(* IEC 61131-3 sources: ECU_Test_Arduino_PLC/PLC_Software, 6 files *)

(* ---- GVL.ST ---- *)
{attribute 'qualified_only'}
VAR_GLOBAL CONSTANT
	uiPeriodcMessageN : UINT := 2;
	uiRXMessageN : UINT := 3;
END_VAR

VAR_GLOBAL
	aPeriodicMessages: ARRAY[1..GVL.uiPeriodcMessageN] OF PERIODIC_MESSAGE;
	aRXMessages: ARRAY[1..GVL.uiRXMessageN] OF RX_MESSAGE;

END_VAR

(* ---- GVL_IO.ST ---- *)
{attribute 'qualified_only'}
VAR_GLOBAL
	//w_CAN_SEND: ARRAY[0..23] OF BYTE;
	//AUX IO
	x_PEDAL_REAL: BOOL;
	x_PEDAL_TYPE: BOOL;

	x_DOG12 : BOOL	;//	J1.E1	Red Changing Light
	x_DOG01	: BOOL	;//	J1.E2	Contactor Supply Control Packs 4-6
	x_DOG02	: BOOL	;//	J1.E3	Contactor Supply Control Packs 7-9
	x_DOG03	: BOOL	;//	J1.E4	Start/Stop Orange LED
	x_DOG04	: BOOL	;//	J1.F1	Start/Stop Green LED
	x_DOG05	: BOOL	;//	J1.F2	Green Charging Light
	x_DOG06	: BOOL	;//	J1.F3 	Contactor Supply Control Packs 1-3
	x_DOG07	: BOOL	;//	J1.F4 	Blue Charging Light
	x_DOG08	: BOOL	;//	J1.G1 	TGC Off Command
	x_DOG09	: BOOL	;//	J1.G2 	TGC On Command
	x_DOG10	: BOOL	;//	J1.G3	LV ePTO Relay Coil control
	x_DOG11	: BOOL	;//	J1.G4	Differential Lock Solenoid LS

	x_DOV01	: BOOL	;//	J1.L1	VCM Wake 1
	x_DOV02	: BOOL	;//	J1.L2	VCM Wake 2
	x_DOV03	: BOOL	;//	J1.L3	VCM Wake 3
	x_DOV04	: BOOL	;//	J1.L4	Governor Valve
	x_DOV05	: BOOL	;//	J1.M1	Regeneration Valve
	x_DOV06	: BOOL	;//	J1.M2	VCM wake 4
	x_DOV07	: BOOL	;//	J1.M3	Auxiliary HVIL Out
	x_DOV08	: BOOL	;//	J1.M4	HV Battery 1-9 Wake

	x_DHLC01 : BOOL	;// J3.21 Cabin Tilt Status [Digital HS-LS Control 1]
	x_DFC01	 : BOOL; // J3.21 Cabin Tilt Status [Digital Float Control 1]
	x_DHLC02 : BOOL	;// J3.22 Drive Req Signal 1 [Digital HS-LS Control 2]
	x_DFC02	 : BOOL; // J3.22 Drive Req Signal 1 [Digital Float Control 2]
	x_DHLC03 : BOOL	;// J3.33 Drive Req Signal 2 [Digital HS-LS Control 3]
	x_DFC03	 : BOOL; // J3.33 Drive Req Signal 2 [Digital Float Control 3]
	x_DHLC04 : BOOL	;// J3.34 Neutral Req Signal [Digital HS-LS Control 4]
	x_DFC04	 : BOOL; // J3.34 Neutral Req Signal [Digital Float Control 4]
	x_DHLC05 : BOOL	;// J3.45 Reverse Req Signal 1 [Digital HS-LS Control 5]
	x_DFC05	 : BOOL; // J3.45 Reverse Req Signal 1 [Digital Float Control 5]
	x_DHLC06 : BOOL	;// J3.46 Reverse Req Signal 2 [Digital HS-LS Control 6]
	x_DFC06	 : BOOL ; // J3.46 Reverse Req Signal 2 [Digital Float Control 6]

	x_CF01	 : BOOL ; // J3.23 Start/Stop Signal 2 [Control Float 1]
	x_CF02	 : BOOL ; // J3.24 Start/Stop Signal 1 [Control Float 2]
	x_CF03	 : BOOL ; // J3.25 APU Sensor Front Signal [Control Float 3]
	x_CF04	 : BOOL ; // J3.26 APU Sensor Rear Signal [Control Float 4]
	x_CF05	 : BOOL ; // J3.27 TGC Off Request [Control Float 5]
	x_CF06	 : BOOL ; // J3.28 TGC On Request [Control Float 6]
	x_CF07	 : BOOL ; // J3.35 FLEX-IN6 [Control Float 7]
	x_CF08	 : BOOL ; // J3.36 FLEX-IN7 [Control Float 8]
	x_CF09	 : BOOL ; // J3.37 FLEX-IN8 [Control Float 9]
	x_CF10	 : BOOL ; // J3.38 Positive Auxiliary Contactor Feedback [Control Float 10]
	x_CF11	 : BOOL ; // J3.39 Negative Auxiliary Contactor Feedback [Control Float 11]
	x_CF12	 : BOOL ; // J3.40 FLEX-IN11 [Control Float 12]
	x_CF13	 : BOOL ; // J3.47 HW E-Stop Signal [Control Float 13]
	x_CF14	 : BOOL ; // J3.48 TPMS Power [Control Float 14]
	x_CF15	 : BOOL ; // J3.49  Differential Lock Sensor Signal [Control Float 15]
	x_CF16	 : BOOL ; // J3.50  Charge Door Position [Control Float 16]

	x_CA01	 : BOOL ; // J3.23 Start/Stop Signal 2 [Control Analog 1]
	x_CA02	 : BOOL ; // J3.24 Start/Stop Signal 1 [Control Analog 2]
	x_CA03	 : BOOL ; // J3.25 APU Sensor Front Signal [Control Analog 3]
	x_CA04	 : BOOL ; // J3.26 APU Sensor Rear Signal [Control Analog 4]
	x_CA05	 : BOOL ; // J3.27 TGC Off Request [Control Analog 5]
	x_CA06	 : BOOL ; // J3.28 TGC On Request [Control Analog 6]
	x_CA07	 : BOOL ; // J3.35 FLEX-IN6 [Control Analog 7]
	x_CA08	 : BOOL ; // J3.36 FLEX-IN7 [Control Analog 8]
	x_CA09	 : BOOL ; // J3.37 FLEX-IN8 [Control Analog 9]
	x_CA10	 : BOOL ; // J3.38 Positive Auxiliary Contactor Feedback [Control Analog 10]
	x_CA11	 : BOOL ; // J3.39 Negative Auxiliary Contactor Feedback [Control Analog 11]
	x_CA12	 : BOOL ; // J3.40 FLEX-IN11 [Control Analog 12]
	x_CA13	 : BOOL ; // J3.47 HW E-Stop Signal [Control Analog 13]
	x_CA14	 : BOOL ; // J3.48 TPMS Power [Control Analog 14]
	x_CA15	 : BOOL ; // J3.49  Differential Lock Sensor Signal [Control Analog 15]
	x_CA16	 : BOOL ; // J3.50  Charge Door Position [Control Analog 16]

	w_FlexIN0	 : WORD ; // J3.23 Start/Stop Signal 2 [FlexIN0]
	w_FlexIN1	 : WORD ; // J3.24 Start/Stop Signal 1 [FlexIN1]
	w_FlexIN2	 : WORD ; // J3.25 APU Sensor Front Signal [FlexIN2]
	w_FlexIN3	 : WORD ; // J3.26 APU Sensor Rear Signal [FlexIN3]
	w_FlexIN4	 : WORD ; // J3.27 TGC Off Request [FlexIN4]
	w_FlexIN5	 : WORD ; // J3.28 TGC On Request [FlexIN5]
	w_FlexIN6	 : WORD ; // J3.35 FLEX-IN6 [FlexIN6]
	w_FlexIN7	 : WORD ; // J3.36 FLEX-IN7 [FlexIN7]
	w_FlexIN8	 : WORD ; // J3.37 FLEX-IN8 [FlexIN8]
	w_FlexIN9	 : WORD ; // J3.38 Positive Auxiliary Contactor Feedback [FlexIN9]
	w_FlexIN10	 : WORD ; // J3.39 Negative Auxiliary Contactor Feedback [FlexIN10]
	w_FlexIN11	 : WORD ; // J3.40 FLEX-IN11 [FlexIN11]
	w_FlexIN12	 : WORD ; // J3.47 HW E-Stop Signal [FlexIN12]
	w_FlexIN13	 : WORD ; // J3.48 TPMS Power [FlexIN13]
	w_FlexIN14	 : WORD ; // J3.49  Differential Lock Sensor Signal [FlexIN14]
	w_FlexIN15	 : WORD ; // J3.50  Charge Door Position [FlexIN15]

	w_AccPedalSig1			: WORD 	;	//J3.8 AccPedalSig1
	w_AccPedalSig2			: WORD  ;	//J3.9 AccPedalSig2
	w_ANC2					: WORD  ;	//J3.10 ANC2
	w_OilLevelSig			: WORD  ;	//J3.11 OilLevelSig
	w_Cabin_Sw_E_Stop_Sig	: WORD  ;	//J3.12 Cabin_Sw_E_Stop_Sig
	w_ANC5					: WORD  ;	//J3.13 ANC5

	b_PWM1_Control_Byte_0	: BYTE ;   // J3.19-20 PWM [Control Byte 0]
	w_PWM1_DO1				: WORD ;   // J3.19 Speed Pulse PWM [DO1]
	w_PWM1_DO2				: WORD ;   // J3.20 Distance Signal [DO2]
	b_PWM1_Control_Byte_2   : BYTE ;  // J3.31-32 PWM [Control Byte 2]
	w_PWM1_DO3				: WORD ;   // J3.31 FLEX_PWM2_NOT_USED [DO3]
	w_PWM1_DO4				: WORD ;   // J3.32 PYRO Crash Event Signal [DO4]

	b_PWM2_Control_Byte_0	: BYTE ;   // J3.43-44 PWM [Control Byte 0]
	w_PWM2_DO1				: WORD ;   // J3.43 FLEX_PWM4 [DO1]
	w_PWM2_DO2				: WORD ;   // J3.44 FLEX_PWM5 [DO2]

//	x_DOV09	: BOOL	;//	X2.28	b
//	x_CrankHSS	: BOOL	;//	X2.36	Cranking Relay HSS
//	x_DOV15	: BOOL	;//	X2.06	Single H out2
//	x_DOV16	: BOOL	;//	X2.04	Single H out1
	//LIN1-GND	: BOOL	;//	X1.05	LIN 1 GND
	x_TRX_P	: BOOL	;//	X1.07	Not Used
	x_TRX_M	: BOOL	;//	X1.08	Not Used
	//x_DIG_ACC_GND: BOOL	;//	X1.09	Accelerator pedal low idle switch
	//x_DIG16	: BOOL	;//	X1.10	PTO 3
	//x_DIG15	: BOOL	;//	X1.11	PTO 2
	//x_DIG14	: BOOL	;//	X1.12	PTO 1
	x_DIB15	: BOOL	;//	X1.13	Hill holder
	x_DIB15H	: BOOL	;//	X1.13	Hill holder
	//LIN2-GND	: BOOL	;//	X1.14	optional
	x_ASG02	: BOOL	;//	X1.15	Accelerator Pedal channel2 Ground
	//CAN6-H	: BOOL	;//	X1.16	Not Used
	//CAN6-L	: BOOL	;//	X1.17	Not Used
	x_ASG01	: BOOL	;//	X1.18	Accelerator Pedal channel1 Ground
	//CAN5-H	: BOOL	;//	X1.19	Body Computer Bus - CAN H
	//CAN5-L	: BOOL	;//	X1.20	Body Computer Bus - CAN L
	w_AI01	: WORD	;//	X1.21	Accelerator Pedal channel 1
	w_AI02	: WORD	;//	X1.22	Accelerator Pedal channel 2
	x_ACC_SW_GND: BOOL	;//	X1.23	Accelerator  pedal low idle switch Ground

	x_ASV01	: BOOL	;//	X1.26	Accelerator Pedal channel 1 Supply
	x_ASV02	: BOOL	;//	X1.27	Accelerator Pedal channel 2 Supply
	x_AWWS_B_In	: BOOL	;//	X1.28	optional
	x_AWWS_B_Out: BOOL	;//	X1.29	optional
	//LIN1-SIG	: BOOL	;//	X1.31	LIN 1 Bus
	//LIN2-SIG	: BOOL	;//	X1.32	optional
	//LIN1-SUP	: BOOL	;//	X1.33	LIN 1 supply
	//LIN2-SUP	: BOOL	;//	X1.34	optional
	x_AWWS_A_In	: BOOL	;//	X1.35	optional
	x_AWWS_A_Out: BOOL	;//	X1.36	optional

	x_TRM_30: BOOL	;//	X2.01	Power Supply
	//CAN9-H	: BOOL	;//	X2.02	optional
	//CAN9-L	: BOOL	;//	X2.03	optional

	x_AI03	: BOOL	;//	X2.07	Analog Input 3
	//x_DIG07	: BOOL	;//	X2.08	Gear High/Low
	x_TRM_15: BOOL	;//	X2.09	Ignition Key
	//CAN1-H	: BOOL	;//	X2.10	Vehicle Data Bus CAN H
	//CAN1-L	: BOOL	;//	X2.11	Vehicle Data Bus CAN L
	//CAN2-H	: BOOL	;//	X2.12	Engine Contro Bus - CAN H
	//CAN2-L	: BOOL	;//	X2.13	Engine Contro Bus - CAN L
	//CAN3-H	: BOOL	;//	X2.14	Expansion Module Bus - CAN H
	//CAN3-L	: BOOL	;//	X2.15	Expansion Module Bus - CAN L
	//CAN4-H	: BOOL	;//	X2.16	ADAS Data Bus CAN FD - CAN H
	//CAN4-L	: BOOL	;//	X2.17	ADAS Data Bus CAN FD - CAN L
	x_TRM_31: BOOL	;//	X2.19	Power Supply GND
	x_DIV04	: BOOL	;//	X2.20	Alcohol Interlock
	//x_DIG12	: BOOL	;//	X2.21	BB Start
	//x_DIG13	: BOOL	;//	X2.22	BB Stop
	//cAN7-H	: BOOL	;//	X2.23	optional
	//CAN7-L	: BOOL	;//	X2.24	optional
	//CAN8-H	: BOOL	;//	X2.25	optional
	//CAN8-L	: BOOL	;//	X2.26	optional

	x_DIB16	: BOOL	;//	X2.30	Halt brake
	x_DIB16H: BOOL	;//	X2.30	Halt brake
	x_DIB17	: BOOL	;//	X2.31	ESP / ASR
	x_DIB17H: BOOL	;//	X2.31	ESP / ASR

	//x_DIG19	: BOOL	;//	X2.34	Clima 22
	//x_DIG18	: BOOL	;//	X2.35	Clima 18

// 	x_DIG01	: BOOL	;//	X3.01	CC Set+
// 	x_DIG02	: BOOL	;//	X3.02	CC Set-
// 	x_DIG03	: BOOL	;//	X3.03	CC Resume
// 	x_DIG04	: BOOL	;//	X3.04	CC Off
	x_DIB05	: BOOL	;//	X3.05	CC GAP-
	x_DIB05H: BOOL	;//	X3.05	CC GAP-
	x_DIB06	: BOOL	;//	X3.06	CC GAP +
	x_DIB06H: BOOL	;//	X3.06	CC GAP +
// 	x_DIG05	: BOOL	;//	X3.07	Ext/Int CC
// 	x_DIG20	: BOOL	;//	X3.08	D/Dm1
// 	x_DIG24	: BOOL	;//	X3.09	R/Rm1
// 	x_DIG22	: BOOL	;//	X3.10	N
// 	x_DIG21	: BOOL	;//	X3.11	D/Dm2
// 	x_DIG25	: BOOL	;//	X3.12	R/Rm2
	x_DIB12	: BOOL	;//	X3.13	Gear Up
	x_DIB12H	: BOOL	;//	X3.13	Gear Up
	x_DIB13	: BOOL	;//	X3.14	Gear Down
	x_DIB13H	: BOOL	;//	X3.14	Gear Down
	x_DIB04	: BOOL	;//	X3.15	FPSL
	x_DIB04H	: BOOL	;//	X3.15	FPSL
	x_DIB02	: BOOL	;//	X3.16	ECO Roll Swt
	x_DIB02H	: BOOL	;//	X3.16	ECO Roll Swt
	x_DIV03	: BOOL	;//	X3.17	Second SL Switch
	x_DIV02	: BOOL	;//	X3.18	Sec. Brake
	x_DIV01	: BOOL	;//	X3.19	Prim. Brake
	x_DIB11	: BOOL	;//	X3.20	ACC
	x_DIB11H	: BOOL	;//	X3.20	ACC
	x_DIB08	: BOOL	;//	X3.21	PECC
	x_DIB08H	: BOOL	;//	X3.21	PECC
	x_DIB01	: BOOL	;//	X3.22	Cranck request (K50)
	x_DIB01H	: BOOL	;//	X3.22	Cranck request (K50)
	x_DIB14	: BOOL	;//	X3.23	Parking Brake Switch
	x_DIB14H	: BOOL	;//	X3.23	Parking Brake Switch
	x_DIG11	: BOOL	;//	X3.24	Cabin Tilt
	x_DIG10	: BOOL	;//	X3.25	Neutral
	x_DIG06	: BOOL	;//	X3.26	Clutch
	//x_DIG17	: BOOL	;//	X3.27	Clutch 2nd
	x_DIB10	: BOOL	;//	X3.28	ABS OFF
	x_DIB10H	: BOOL	;//	X3.28	ABS OFF
	//x_DIG09	: BOOL	;//	X3.29	EB Mode 1
	x_DIB07	: BOOL	;//	X3.30	EB request
	x_DIB07H	: BOOL	;//	X3.30	EB request
	//x_DIG27	: BOOL	;//	X3.31	CSF - LDWS
	//x_DIG23	: BOOL	;//	X3.32	Heavy Offroad
	x_DIB03	: BOOL	;//	X3.33	Rocking Mode
	x_DIB03H	: BOOL	;//	X3.33	Rocking Mode
	x_DIB09	: BOOL	;//	X3.34	 Power mode
	x_DIB09H	: BOOL	;//	X3.34	 Power mode
	//x_DIG26	: BOOL	;//	X3.35	Silent Mode
	//x_DIG08	: BOOL	;//	X3.36	ECO Mode
END_VAR

(* ---- FB_RXCanMessageelaboration.ST ---- *)
FUNCTION_BLOCK FB_RXCanMessageElaboration
VAR_INPUT
	wRxId:WORD;
	bRxNBytes:BYTE;
	aRxBuffer: ARRAY [0..7] OF BYTE;
END_VAR
VAR_OUTPUT
END_VAR
VAR
	_FbCanTx11BitFrame : FbCanTx11BitFrame;
	xCANTxTrigger : BOOL;
	lut1,lut2: LUT;
END_VAR

xCANTxTrigger := FALSE;//no answer required

CASE wRxId OF
// 	16#75C:
// 			//ON MESSAGE ACTION
// 			IF aRxBuffer[0] = 0 THEN
// 				GVL.DO01 := FALSE;
// 			ELSE
// 				GVL.DO01 := TRUE;
// 			END_IF
// 			xCANTxTrigger := TRUE;
	16#11://BANCO_VCM4_Command
			GVL_IO.x_PEDAL_TYPE := aRxBuffer[0].0;//Pedal_Type
			GVL_IO.x_TRM_30 := aRxBuffer[0].1;//Power_Supply
			GVL_IO.x_TRM_15 := aRxBuffer[0].2;//Ignition_Key
			GVL_IO.x_PEDAL_REAL	:= aRxBuffer[0].3;//Accelerator_Pedal

	16#12://BANCO_VCM4_ANALOG_Critical_ADC (597_3) ++
			//ON MESSAGE ACTION
			GVL_IO.w_AccPedalSig1 := INT_TO_WORD(REAL_TO_INT((WORD_TO_REAL(SHL(BYTE_TO_WORD(aRxBuffer[1]),8) + BYTE_TO_WORD(aRxBuffer[0]))) * 0.001 * 32767) ); // Refer to the manual of 597 page 34
			GVL_IO.w_AccPedalSig2 := INT_TO_WORD(REAL_TO_INT((WORD_TO_REAL(SHL(BYTE_TO_WORD(aRxBuffer[3]),8) + BYTE_TO_WORD(aRxBuffer[2]))) * 0.001 * 32767) ); // Refer to the manual of 597 page 34
			GVL_IO.w_OilLevelSig := INT_TO_WORD(REAL_TO_INT((WORD_TO_REAL(SHL(BYTE_TO_WORD(aRxBuffer[5]),8) + BYTE_TO_WORD(aRxBuffer[4]))) * 0.001 * 32767) ); // Refer to the manual of 597 page 34
			GVL_IO.w_Cabin_Sw_E_Stop_Sig := INT_TO_WORD(REAL_TO_INT((WORD_TO_REAL(SHL(BYTE_TO_WORD(aRxBuffer[7]),8) + BYTE_TO_WORD(aRxBuffer[6]))) * 0.001 * 32767) ); // Refer to the manual of 597 page 34

	16#14://BANCO_VCM4_DI ++
			GVL_IO.x_DHLC01 := aRxBuffer[0].0; // Cabin_Tilt_Status_HS_LS
			GVL_IO.x_DFC01  := aRxBuffer[0].1; // Cabin_Tilt_Status_Float
			GVL_IO.x_DHLC02 := aRxBuffer[0].2; // Drive_Req_Signal_1_HS_LS
			GVL_IO.x_DFC02  := aRxBuffer[0].3; // Drive_Req_Signal_1_Float
			GVL_IO.x_DHLC03 := aRxBuffer[0].4; // Drive_Req_Signal_2_HS_LS
			GVL_IO.x_DFC03  := aRxBuffer[0].5; // Drive_Req_Signal_2_Float
			GVL_IO.x_DHLC04 := aRxBuffer[0].6; // Neutral_Req_Signal_HS_LS
			GVL_IO.x_DFC04  := aRxBuffer[0].7; // Neutral_Req_Signal_Float
			GVL_IO.x_DHLC05 := aRxBuffer[1].0; // Reverse_Req_Signal_1_HS_LS
			GVL_IO.x_DFC05  := aRxBuffer[1].1; // Reverse_Req_Signal_1_Float
			GVL_IO.x_DHLC06 := aRxBuffer[1].2; // Reverse_Req_Signal_2_HS_LS
			GVL_IO.x_DFC06  := aRxBuffer[1].3; // Reverse_Req_Signal_2_Float
			GVL_IO.x_DIB05  := aRxBuffer[1].4; // Power_Control
			GVL_IO.x_DIB05H := aRxBuffer[1].5; // K15-Ignition-Control

// 	16#15://BANCO_VCM4_PWM_IN ++
// 			GVL_IO.b_PWM1_Control_Byte_0 :=  aRxBuffer[0];
// 			GVL_IO.b_PWM1_Control_Byte_2 :=  aRxBuffer[1];
// 			GVL_IO.w_PWM1_DO1 := REAL_TO_WORD((WORD_TO_REAL(SHL(BYTE_TO_WORD(aRxBuffer[3]),8) + BYTE_TO_WORD(aRxBuffer[2]))));
// 			GVL_IO.w_PWM1_DO2 := REAL_TO_WORD((WORD_TO_REAL(SHL(BYTE_TO_WORD(aRxBuffer[5]),8) + BYTE_TO_WORD(aRxBuffer[4]))));
// 			GVL_IO.w_PWM1_DO4 := REAL_TO_WORD((WORD_TO_REAL(SHL(BYTE_TO_WORD(aRxBuffer[7]),8) + BYTE_TO_WORD(aRxBuffer[6]))));

	16#16://BANCO_VCM4_Analog_Control ++
			GVL_IO.x_CF01 := aRxBuffer[0].0;//Start_Stop_Signal_2_Float 0
			GVL_IO.x_CA01 := aRxBuffer[0].1;//Start_Stop_Signal_2_Analog 0
			GVL_IO.x_CF02 := aRxBuffer[0].2;//Start_Stop_Signal_1_Float 1
			GVL_IO.x_CA02 := aRxBuffer[0].3;//Start_Stop_Signal_1_Analog 1
			GVL_IO.x_CF03 := aRxBuffer[0].4;//APU_Sensor_Front_Signal_Float 2
			GVL_IO.x_CA03 := aRxBuffer[0].5;//APU_Sensor_Front_Signal_Analog 2
			GVL_IO.x_CF04 := aRxBuffer[0].6;//APU_Sensor_Rear_Signal_Float 3
			GVL_IO.x_CA04 := aRxBuffer[0].7;//APU_Sensor_Rear_Signal_Analog 3
			GVL_IO.x_CF05 := aRxBuffer[1].0;//TGC_Off_Request_Float 4
			GVL_IO.x_CA05 := aRxBuffer[1].1;//TGC_Off_Request_Analog 4
			GVL_IO.x_CF06 := aRxBuffer[1].2;//TGC_On_Request_Float 5
			GVL_IO.x_CA06 := aRxBuffer[1].3;//TGC_On_Request_Analog 5
			GVL_IO.x_CF07 := aRxBuffer[1].4;//Not_Used_FLEX_IN6_Float 6
			GVL_IO.x_CA07 := aRxBuffer[1].5;//Not_Used_FLEX_IN6_Analog 6
			GVL_IO.x_CF08 := aRxBuffer[1].6;//Not_Used_FLEX_IN7_Float 7
			GVL_IO.x_CA08 := aRxBuffer[1].7;//Not_Used_FLEX_IN7_Analog 7
			GVL_IO.x_CF09 := aRxBuffer[2].0;//Not_Used_FLEX_IN8_Float 8
			GVL_IO.x_CA09 := aRxBuffer[2].1;//Not_Used_FLEX_IN8_Analog 8
			GVL_IO.x_CF10 := aRxBuffer[2].2;//Positive_Auxiliary_Contactor_Feedback_Float 9
			GVL_IO.x_CA10 := aRxBuffer[2].3;//Positive_Auxiliary_Contactor_Feedback_Analog 9
			GVL_IO.x_CF11 := aRxBuffer[2].4;//Negative_Auxiliary_Contactor_Feedback_Float 10
			GVL_IO.x_CA11 := aRxBuffer[2].5;//Negative_Auxiliary_Contactor_Feedback_Analog 10
			GVL_IO.x_CF12 := aRxBuffer[2].6;//Not_Used_FLEX_IN11_Float 11
			GVL_IO.x_CA12 := aRxBuffer[2].7;//Not_Used_FLEX_IN11_Analog 11
			GVL_IO.x_CF13 := aRxBuffer[3].0;//HW_E_Stop_Signal_Float 12
			GVL_IO.x_CA13 := aRxBuffer[3].1;//HW_E_Stop_Signal_Analog 12
			GVL_IO.x_CF14 := aRxBuffer[3].2;//TPMS_Power_Float 13
			GVL_IO.x_CA14 := aRxBuffer[3].3;//TPMS_Power_Analog 13
			GVL_IO.x_CF15 := aRxBuffer[3].4;//Differential_Lock_Sensor_Signal_Float 14
			GVL_IO.x_CA15 := aRxBuffer[3].5;//Differential_Lock_Sensor_Signal_Analog 14
			GVL_IO.x_CF16 := aRxBuffer[3].6;//Charge_Door_Position_Float 15
			GVL_IO.x_CA16 := aRxBuffer[3].7;//Charge_Door_Position_Analog 15

// /// Arduino ///
// 		16#18: //BANCO_VCM4_PWM_HBO_0
// 		16#19: //BANCO_VCM4_PWM_HBO_1
// 		16#1A: //BANCO_VCM4_PWM_HBO_2
// 		16#1B: //BANCO_VCM4_PWM_HBO_3

		16#1C: //BANCO_VCM4_Analog_IN_0_3 ++
			GVL_IO.w_FlexIN0 := INT_TO_WORD(REAL_TO_INT((WORD_TO_REAL(SHL(BYTE_TO_WORD(aRxBuffer[1]),8) + BYTE_TO_WORD(aRxBuffer[0]))) * 0.001 * 32767) ); // Refer to the manual of 597 page 34
			GVL_IO.w_FlexIN1 := INT_TO_WORD(REAL_TO_INT((WORD_TO_REAL(SHL(BYTE_TO_WORD(aRxBuffer[3]),8) + BYTE_TO_WORD(aRxBuffer[2]))) * 0.001 * 32767) );
			GVL_IO.w_FlexIN2 := INT_TO_WORD(REAL_TO_INT((WORD_TO_REAL(SHL(BYTE_TO_WORD(aRxBuffer[5]),8) + BYTE_TO_WORD(aRxBuffer[4]))) * 0.001 * 32767) );
			GVL_IO.w_FlexIN3 := INT_TO_WORD(REAL_TO_INT((WORD_TO_REAL(SHL(BYTE_TO_WORD(aRxBuffer[7]),8) + BYTE_TO_WORD(aRxBuffer[6]))) * 0.001 * 32767) );
		16#1D: //BANCO_VCM4_Analog_IN_4_7 ++
			GVL_IO.w_FlexIN4 := INT_TO_WORD(REAL_TO_INT((WORD_TO_REAL(SHL(BYTE_TO_WORD(aRxBuffer[1]),8) + BYTE_TO_WORD(aRxBuffer[0]))) * 0.001 * 32767) );
			GVL_IO.w_FlexIN5 := INT_TO_WORD(REAL_TO_INT((WORD_TO_REAL(SHL(BYTE_TO_WORD(aRxBuffer[3]),8) + BYTE_TO_WORD(aRxBuffer[2]))) * 0.001 * 32767) );
			GVL_IO.w_FlexIN6 := INT_TO_WORD(REAL_TO_INT((WORD_TO_REAL(SHL(BYTE_TO_WORD(aRxBuffer[5]),8) + BYTE_TO_WORD(aRxBuffer[4]))) * 0.001 * 32767) );
			GVL_IO.w_FlexIN7 := INT_TO_WORD(REAL_TO_INT((WORD_TO_REAL(SHL(BYTE_TO_WORD(aRxBuffer[7]),8) + BYTE_TO_WORD(aRxBuffer[6]))) * 0.001 * 32767) );
		16#1E: //BANCO_VCM4_Analog_IN_8_11 ++
			GVL_IO.w_FlexIN8 := INT_TO_WORD(REAL_TO_INT((WORD_TO_REAL(SHL(BYTE_TO_WORD(aRxBuffer[1]),8) + BYTE_TO_WORD(aRxBuffer[0]))) * 0.001 * 32767) );
			GVL_IO.w_FlexIN9 := INT_TO_WORD(REAL_TO_INT((WORD_TO_REAL(SHL(BYTE_TO_WORD(aRxBuffer[3]),8) + BYTE_TO_WORD(aRxBuffer[2]))) * 0.001 * 32767) );
			GVL_IO.w_FlexIN10 := INT_TO_WORD(REAL_TO_INT((WORD_TO_REAL(SHL(BYTE_TO_WORD(aRxBuffer[5]),8) + BYTE_TO_WORD(aRxBuffer[4]))) * 0.001 * 32767) );
			GVL_IO.w_FlexIN11 := INT_TO_WORD(REAL_TO_INT((WORD_TO_REAL(SHL(BYTE_TO_WORD(aRxBuffer[7]),8) + BYTE_TO_WORD(aRxBuffer[6]))) * 0.001 * 32767) );
		16#1F: //BANCO_VCM4_Analog_IN_12_15 ++
			GVL_IO.w_FlexIN12 := INT_TO_WORD(REAL_TO_INT((WORD_TO_REAL(SHL(BYTE_TO_WORD(aRxBuffer[1]),8) + BYTE_TO_WORD(aRxBuffer[0]))) * 0.001 * 32767) );
			GVL_IO.w_FlexIN13 := INT_TO_WORD(REAL_TO_INT((WORD_TO_REAL(SHL(BYTE_TO_WORD(aRxBuffer[3]),8) + BYTE_TO_WORD(aRxBuffer[2]))) * 0.001 * 32767) );
			GVL_IO.w_FlexIN14 := INT_TO_WORD(REAL_TO_INT((WORD_TO_REAL(SHL(BYTE_TO_WORD(aRxBuffer[5]),8) + BYTE_TO_WORD(aRxBuffer[4]))) * 0.001 * 32767) );
			GVL_IO.w_FlexIN15 := INT_TO_WORD(REAL_TO_INT((WORD_TO_REAL(SHL(BYTE_TO_WORD(aRxBuffer[7]),8) + BYTE_TO_WORD(aRxBuffer[6]))) * 0.001 * 32767) );

// 		16#20: //BANCO_VCM4_PWM_IN_NOT_USED ++
// 			GVL_IO.b_PWM1_Control_Byte_2 :=  aRxBuffer[0];
// 			GVL_IO.b_PWM2_Control_Byte_0 :=  aRxBuffer[1];
// 			GVL_IO.w_PWM1_DO3 := REAL_TO_WORD((WORD_TO_REAL(SHL(BYTE_TO_WORD(aRxBuffer[3]),8) + BYTE_TO_WORD(aRxBuffer[2]))));
// 			GVL_IO.w_PWM2_DO1 := REAL_TO_WORD((WORD_TO_REAL(SHL(BYTE_TO_WORD(aRxBuffer[5]),8) + BYTE_TO_WORD(aRxBuffer[4]))));
// 			GVL_IO.w_PWM2_DO2 := REAL_TO_WORD((WORD_TO_REAL(SHL(BYTE_TO_WORD(aRxBuffer[7]),8) + BYTE_TO_WORD(aRxBuffer[6]))));

		16#21: //BANCO_VCM4_Analog_Critical_ADC_NOT_USED ++
			GVL_IO.w_ANC2 := INT_TO_WORD(REAL_TO_INT((WORD_TO_REAL(SHL(BYTE_TO_WORD(aRxBuffer[1]),8) + BYTE_TO_WORD(aRxBuffer[0]))) * 0.001 * 32767) );
			GVL_IO.w_ANC5 := INT_TO_WORD(REAL_TO_INT((WORD_TO_REAL(SHL(BYTE_TO_WORD(aRxBuffer[3]),8) + BYTE_TO_WORD(aRxBuffer[2]))) * 0.001 * 32767) );
END_CASE

//ON MESSAGE ANSWER
_FbCanTx11BitFrame( xEnable := TRUE,
					I_Port := CAN_Gateway,
					wCanId := 16#75D,
					xRtrFrame := FALSE,
					aTxBuffer := aRxBuffer,
					bTxNBytes := bRxNBytes,
					xTxTrigger := xCANTxTrigger,
					xValid =>,
					xError =>,
					xBusy =>,
					oStatus =>
					);

(* ---- PLC_INPUT.ST ---- *)
PROGRAM PLC_INPUT
VAR
	x_i_1405_1_1	AT	%IX26.0	:	BOOL	;
	x_i_1405_1_2	AT	%IX26.1	:	BOOL	;
	x_i_1405_1_3	AT	%IX26.2	:	BOOL	;
	x_i_1405_1_4	AT	%IX26.3	:	BOOL	;
	x_i_1405_1_5	AT	%IX26.4	:	BOOL	;
	x_i_1405_1_6	AT	%IX26.5	:	BOOL	;
	x_i_1405_1_7	AT	%IX26.6	:	BOOL	;
	x_i_1405_1_8	AT	%IX26.7	:	BOOL	;
	x_i_1405_1_9	AT	%IX26.8	:	BOOL	;
	x_i_1405_1_10	AT	%IX26.9	:	BOOL	;
	x_i_1405_1_11	AT	%IX26.10:	BOOL	;
	x_i_1405_1_12	AT	%IX26.11:	BOOL	;
	x_i_1405_1_13	AT	%IX26.12:	BOOL	;
	x_i_1405_1_14	AT	%IX26.13:	BOOL	;
	x_i_1405_1_15	AT	%IX26.14:	BOOL	;
	x_i_1405_1_16	AT	%IX26.15:	BOOL	;

	x_i_1407_1_1	AT	%IX28.0	:	BOOL	;
	x_i_1407_1_2	AT	%IX28.1	:	BOOL	;
	x_i_1407_1_3	AT	%IX28.2	:	BOOL	;
	x_i_1407_1_4	AT	%IX28.3	:	BOOL	;
	x_i_1407_1_5	AT	%IX28.4	:	BOOL	;
	x_i_1407_1_6	AT	%IX28.5	:	BOOL	;
	x_i_1407_1_7	AT	%IX28.6	:	BOOL	;
	x_i_1407_1_8	AT	%IX28.7	:	BOOL	;
	x_i_1407_1_9	AT	%IX28.8	:	BOOL	;
	x_i_1407_1_10	AT	%IX28.9	:	BOOL	;
	x_i_1407_1_11	AT	%IX28.10:	BOOL	;
	x_i_1407_1_12	AT	%IX28.11:	BOOL	;
	x_i_1407_1_13	AT	%IX28.12:	BOOL	;
	x_i_1407_1_14	AT	%IX28.13:	BOOL	;
	x_i_1407_1_15	AT	%IX28.14:	BOOL	;
	x_i_1407_1_16	AT	%IX28.15:	BOOL	;

END_VAR

GVL_IO.x_DOV01	:=	x_i_1405_1_1;
GVL_IO.x_DOV02	:=	x_i_1405_1_2;
GVL_IO.x_DOV03	:=	x_i_1405_1_3;
GVL_IO.x_DOV04	:=	x_i_1405_1_4;
GVL_IO.x_DOV05	:=	x_i_1405_1_5;
GVL_IO.x_DOV06	:=	x_i_1405_1_6;
GVL_IO.x_DOV07	:=	x_i_1405_1_7;
GVL_IO.x_DOV08	:=	x_i_1405_1_8;
//GVL_IO.x_DOV09	:=	x_i_1405_1_9;
//GVL_IO.x_CrankHSS:=	x_i_1405_1_10;
//GVL_IO.	:=	x_i_1405_1_11	;
//GVL_IO.	:=	x_i_1405_1_12	;
//GVL_IO.	:=	x_i_1405_1_13	;
//GVL_IO.	:=	x_i_1405_1_14	;
//GVL_IO.x_DOV15	:=	x_i_1405_1_15;//single H out 2
//GVL_IO.x_DOV16	:=	x_i_1405_1_16;

GVL_IO.x_DOG01	:=	x_i_1407_1_1	;
GVL_IO.x_DOG02	:=	x_i_1407_1_2	;
GVL_IO.x_DOG03	:=	x_i_1407_1_3	;
GVL_IO.x_DOG04	:=	x_i_1407_1_4	;
GVL_IO.x_DOG05  :=	x_i_1407_1_5	;
GVL_IO.x_DOG06  :=	x_i_1407_1_6	;
GVL_IO.x_DOG07	:=	x_i_1407_1_7	;
GVL_IO.x_DOG08	:=	x_i_1407_1_8	;
GVL_IO.x_DOG09	:=	x_i_1407_1_9	;
GVL_IO.x_DOG10	:=	x_i_1407_1_10	;
GVL_IO.x_DOG11	:=	x_i_1407_1_11	;
GVL_IO.x_DOG12	:=	x_i_1407_1_12	;
//GVL_IO.	:=	x_i_1407_1_13	;
//GVL_IO.	:=	x_i_1407_1_14	;
//GVL_IO.	:=	x_i_1407_1_15	;
//GVL_IO.	:=	x_i_1407_1_16	;

(* ---- PLC_OUTPUT.ST ---- *)
PROGRAM PLC_OUTPUT
VAR
	//w_q_658_1		AT  %QB0	:   ARRAY[0..23] OF BYTE;
	x_q_1504_1_1	AT	%QX24.0	:	BOOL	;
	x_q_1504_1_2	AT	%QX24.1	:	BOOL	;
	x_q_1504_1_3	AT	%QX24.2	:	BOOL	;
	x_q_1504_1_4	AT	%QX24.3	:	BOOL	;
	x_q_1504_1_5	AT	%QX24.4	:	BOOL	;
	x_q_1504_1_6	AT	%QX24.5	:	BOOL	;
	x_q_1504_1_7	AT	%QX24.6	:	BOOL	;
	x_q_1504_1_8	AT	%QX24.7	:	BOOL	;
	x_q_1504_1_9	AT	%QX24.8	:	BOOL	;
	x_q_1504_1_10	AT	%QX24.9	:	BOOL	;
	x_q_1504_1_11	AT	%QX24.10:	BOOL	;
	x_q_1504_1_12	AT	%QX24.11:	BOOL	;
	x_q_1504_1_13	AT	%QX24.12:	BOOL	;
	x_q_1504_1_14	AT	%QX24.13:	BOOL	;
	x_q_1504_1_15	AT	%QX24.14:	BOOL	;
	x_q_1504_1_16	AT	%QX24.15:	BOOL	;

	x_q_1504_2_1	AT	%QX26.0	:	BOOL	;
	x_q_1504_2_2	AT	%QX26.1	:	BOOL	;
	x_q_1504_2_3	AT	%QX26.2	:	BOOL	;
	x_q_1504_2_4	AT	%QX26.3	:	BOOL	;
	x_q_1504_2_5	AT	%QX26.4	:	BOOL	;
	x_q_1504_2_6	AT	%QX26.5	:	BOOL	;
	x_q_1504_2_7	AT	%QX26.6	:	BOOL	;
	x_q_1504_2_8	AT	%QX26.7	:	BOOL	;
	x_q_1504_2_9	AT	%QX26.8	:	BOOL	;
	x_q_1504_2_10	AT	%QX26.9	:	BOOL	;
	x_q_1504_2_11	AT	%QX26.10:	BOOL	;
	x_q_1504_2_12	AT	%QX26.11:	BOOL	;
	x_q_1504_2_13	AT	%QX26.12:	BOOL	;
	x_q_1504_2_14	AT	%QX26.13:	BOOL	;
	x_q_1504_2_15	AT	%QX26.14:	BOOL	;
	x_q_1504_2_16	AT	%QX26.15:	BOOL	;

	x_q_1504_3_1	AT	%QX28.0	:	BOOL	;
	x_q_1504_3_2	AT	%QX28.1	:	BOOL	;
	x_q_1504_3_3	AT	%QX28.2	:	BOOL	;
	x_q_1504_3_4	AT	%QX28.3	:	BOOL	;
	x_q_1504_3_5	AT	%QX28.4	:	BOOL	;
	x_q_1504_3_6	AT	%QX28.5	:	BOOL	;
	x_q_1504_3_7	AT	%QX28.6	:	BOOL	;
	x_q_1504_3_8	AT	%QX28.7	:	BOOL	;
	x_q_1504_3_9	AT	%QX28.8	:	BOOL	;
	x_q_1504_3_10	AT	%QX28.9	:	BOOL	;
	x_q_1504_3_11	AT	%QX28.10:	BOOL	;
	x_q_1504_3_12	AT	%QX28.11:	BOOL	;
	x_q_1504_3_13	AT	%QX28.12:	BOOL	;
	x_q_1504_3_14	AT	%QX28.13:	BOOL	;
	x_q_1504_3_15	AT	%QX28.14:	BOOL	;
	x_q_1504_3_16	AT	%QX28.15:	BOOL	;

	w_q_597_1_1	AT	%QW15	:	WORD	;
	w_q_597_1_2	AT	%QW16	:	WORD	;
	w_q_597_1_3	AT	%QW17	:	WORD	;
	w_q_597_1_4	AT	%QW18	:	WORD	;
	w_q_597_1_5	AT	%QW19	:	WORD	;
	w_q_597_1_6	AT	%QW20	:	WORD	;
	w_q_597_1_7	AT	%QW21	:	WORD	;
	w_q_597_1_8	AT	%QW22	:	WORD	;

	w_q_597_2_1	AT	%QW23	:	WORD	;
	w_q_597_2_2	AT	%QW24	:	WORD	;
	w_q_597_2_3	AT	%QW25	:	WORD	;
	w_q_597_2_4	AT	%QW26	:	WORD	;
	w_q_597_2_5	AT	%QW27	:	WORD	;
	w_q_597_2_6	AT	%QW28	:	WORD	;
	w_q_597_2_7	AT	%QW29	:	WORD	;
	w_q_597_2_8	AT	%QW30	:	WORD	;

	w_q_597_3_1	AT	%QW31	:	WORD	;
	w_q_597_3_2	AT	%QW32	:	WORD	;
	w_q_597_3_3	AT	%QW33	:	WORD	;
	w_q_597_3_4	AT	%QW34	:	WORD	;
	w_q_597_3_5	AT	%QW35	:	WORD	;
	w_q_597_3_6	AT	%QW36	:	WORD	;

	b_q_677_1_1 AT  %QB78	:	BYTE	; //Control Byte 1
	w_q_677_1_2 AT  %QW40	:	WORD	; // DO1
	//b_q_677_1_3 AT  %QB82	:	BYTE	; //Control Byte 2
	w_q_677_1_4 AT  %QW42	:	WORD	; // DO2
	b_q_677_1_5 AT  %QB86	:	BYTE	; //Control Byte 3
	//w_q_677_1_6 AT  %QW44	:	WORD	; // DO3
	//b_q_677_1_7 AT  %QB90	:	BYTE	; //Control Byte 4
	w_q_677_1_8 AT  %QW46	:	WORD	; // DO4

	b_q_677_2_1 AT  %QB94	:	BYTE	; //Control Byte 1
	w_q_677_2_2 AT  %QW48	:	WORD	; // DO1
	//b_q_677_2_3 AT  %QB98	:	BYTE	; //Control Byte 2
	w_q_677_2_4 AT  %QW50	:	WORD	; // DO2
	//b_q_677_2_5 AT  %QB102	:	BYTE	; //Control Byte 3
	//w_q_677_2_6 AT  %QW52	:	WORD	; // DO3
	//b_q_677_2_7 AT  %QB106	:	BYTE	; //Control Byte 4
	//w_q_677_2_8 AT  %QW54	:	WORD	; // DO4

// 	x_q_1505_1_1	AT	%QX30.0	:	BOOL	;
// 	x_q_1505_1_2	AT	%QX30.1	:	BOOL	;
// 	x_q_1505_1_3	AT	%QX30.2	:	BOOL	;
// 	x_q_1505_1_4	AT	%QX30.3	:	BOOL	;
// 	x_q_1505_1_5	AT	%QX30.4	:	BOOL	;
// 	x_q_1505_1_6	AT	%QX30.5	:	BOOL	;
// 	x_q_1505_1_7	AT	%QX30.6	:	BOOL	;
// 	x_q_1505_1_8	AT	%QX30.7	:	BOOL	;
// 	x_q_1505_1_9	AT	%QX30.8	:	BOOL	;
// 	x_q_1505_1_10	AT	%QX30.9	:	BOOL	;
// 	x_q_1505_1_11	AT	%QX30.10:	BOOL	;
// 	x_q_1505_1_12	AT	%QX30.11:	BOOL	;
// 	x_q_1505_1_13	AT	%QX30.12:	BOOL	;
// 	x_q_1505_1_14	AT	%QX30.13:	BOOL	;
// 	x_q_1505_1_15	AT	%QX30.14:	BOOL	;
// 	x_q_1505_1_16	AT	%QX30.15:	BOOL	;
//
// 	x_q_1505_2_1	AT	%QX32.0	:	BOOL	;
// 	x_q_1505_2_2	AT	%QX32.1	:	BOOL	;
// 	x_q_1505_2_3	AT	%QX32.2	:	BOOL	;
// 	x_q_1505_2_4	AT	%QX32.3	:	BOOL	;
// 	x_q_1505_2_5	AT	%QX32.4	:	BOOL	;
// 	x_q_1505_2_6	AT	%QX32.5	:	BOOL	;
// 	x_q_1505_2_7	AT	%QX32.6	:	BOOL	;
// 	x_q_1505_2_8	AT	%QX32.7	:	BOOL	;
// 	x_q_1505_2_9	AT	%QX32.8	:	BOOL	;
// 	x_q_1505_2_10	AT	%QX32.9	:	BOOL	;
// 	x_q_1505_2_11	AT	%QX32.10:	BOOL	;
// 	x_q_1505_2_12	AT	%QX32.11:	BOOL	;
// 	x_q_1505_2_13	AT	%QX32.12:	BOOL	;
// 	x_q_1505_2_14	AT	%QX32.13:	BOOL	;
// 	x_q_1505_2_15	AT	%QX32.14:	BOOL	;
// 	x_q_1505_2_16	AT	%QX32.15:	BOOL	;
//
// 	w_q_550_1_1		AT %QW17: WORD;
// 	w_q_550_1_2		AT %QW18: WORD;
// 	//w_q_559_1_3		AT %QW17: WORD;
// 	//w_q_559_1_4		AT %QW17: WORD;

END_VAR

//w_q_658_1		:=	GVL_IO.w_CAN_SEND;

x_q_1504_1_1	:=	GVL_IO.x_DHLC01	;
x_q_1504_1_2	:=	GVL_IO.x_DFC01	;
x_q_1504_1_3	:=	GVL_IO.x_DHLC02	;
x_q_1504_1_4	:=	GVL_IO.x_DFC02;
x_q_1504_1_5	:=	GVL_IO.x_DHLC03	;
x_q_1504_1_6	:=	GVL_IO.x_DFC03;
x_q_1504_1_7	:=	GVL_IO.x_DHLC04;
x_q_1504_1_8	:=	GVL_IO.x_DFC04;
x_q_1504_1_9	:=	GVL_IO.x_DHLC05;
x_q_1504_1_10	:=	GVL_IO.x_DFC05	;
x_q_1504_1_11	:=	GVL_IO.x_DHLC06;
x_q_1504_1_12	:=	GVL_IO.x_DFC06	;
x_q_1504_1_13	:=	GVL_IO.x_DIB05;
x_q_1504_1_14	:=	GVL_IO.x_DIB05H	;
//x_q_1504_1_15	:=	GVL_IO.x_DIB06;
//x_q_1504_1_16	:=	GVL_IO.x_DIB06H	;

x_q_1504_2_1	:=	GVL_IO.x_CF01	;
x_q_1504_2_2	:=	GVL_IO.x_CF02	;
x_q_1504_2_3	:=	GVL_IO.x_CF03	;
x_q_1504_2_4	:=	GVL_IO.x_CF04	;
x_q_1504_2_5	:=	GVL_IO.x_CF05	;
x_q_1504_2_6	:=	GVL_IO.x_CF06	;
x_q_1504_2_7	:=	GVL_IO.x_CF07	;
x_q_1504_2_8	:=	GVL_IO.x_CF08	;
x_q_1504_2_9	:=	GVL_IO.x_CF09	;
x_q_1504_2_10	:=	GVL_IO.x_CF10	;
x_q_1504_2_11	:=	GVL_IO.x_CF11	;
x_q_1504_2_12	:=	GVL_IO.x_CF12	;
x_q_1504_2_13	:=	GVL_IO.x_CF13	;
x_q_1504_2_14	:=	GVL_IO.x_CF14	;
x_q_1504_2_15	:=	GVL_IO.x_CF15	;
x_q_1504_2_16	:=	GVL_IO.x_CF16	;

x_q_1504_3_1	:=	GVL_IO.x_CA01	;
x_q_1504_3_2	:=	GVL_IO.x_CA02	;
x_q_1504_3_3	:=	GVL_IO.x_CA03	;
x_q_1504_3_4	:=	GVL_IO.x_CA04	;
x_q_1504_3_5	:=	GVL_IO.x_CA05	;
x_q_1504_3_6	:=	GVL_IO.x_CA06	;
x_q_1504_3_7	:=	GVL_IO.x_CA07	;
x_q_1504_3_8	:=	GVL_IO.x_CA08	;
x_q_1504_3_9	:=	GVL_IO.x_CA09	;
x_q_1504_3_10	:=	GVL_IO.x_CA10	;
x_q_1504_3_11	:=	GVL_IO.x_CA11	;
x_q_1504_3_12	:=	GVL_IO.x_CA12	;
x_q_1504_3_13	:=	GVL_IO.x_CA13	;
x_q_1504_3_14	:=	GVL_IO.x_CA14	;//alco
x_q_1504_3_15	:=	GVL_IO.x_CA15	;
x_q_1504_3_16	:=	GVL_IO.x_CA16	;

w_q_597_1_1		:=	GVL_IO.w_FlexIN0 ;
w_q_597_1_2		:=	GVL_IO.w_FlexIN1 ;
w_q_597_1_3		:=	GVL_IO.w_FlexIN2 ;
w_q_597_1_4		:=	GVL_IO.w_FlexIN3 ;
w_q_597_1_5		:=	GVL_IO.w_FlexIN4 ;
w_q_597_1_6		:=	GVL_IO.w_FlexIN5 ;
w_q_597_1_7		:=	GVL_IO.w_FlexIN6 ;
w_q_597_1_8		:=	GVL_IO.w_FlexIN7 ;

w_q_597_2_1		:=	GVL_IO.w_FlexIN8 ;
w_q_597_2_2		:=	GVL_IO.w_FlexIN9 ;
w_q_597_2_3		:=	GVL_IO.w_FlexIN10 ;
w_q_597_2_4		:=	GVL_IO.w_FlexIN11 ;
w_q_597_2_5		:=	GVL_IO.w_FlexIN12 ;
w_q_597_2_6		:=	GVL_IO.w_FlexIN13 ;
w_q_597_2_7		:=	GVL_IO.w_FlexIN14 ;
w_q_597_2_8		:=	GVL_IO.w_FlexIN15 ;

w_q_597_3_1		:=	GVL_IO.w_AccPedalSig1 ;
w_q_597_3_2		:=	GVL_IO.w_AccPedalSig2 ;
w_q_597_3_3		:=	GVL_IO.w_ANC2 ;
w_q_597_3_4		:=	GVL_IO.w_OilLevelSig ;
w_q_597_3_5		:=	GVL_IO.w_Cabin_Sw_E_Stop_Sig ;
w_q_597_3_6		:=	GVL_IO.w_ANC5 ;

b_q_677_1_1		:=	GVL_IO.b_PWM1_Control_Byte_0	;
w_q_677_1_2		:=	GVL_IO.w_PWM1_DO1;
//b_q_677_1_3		:=	GVL_IO.b_PWM1_Control_Byte_1	;
w_q_677_1_4		:=	GVL_IO.w_PWM1_DO2 ;
b_q_677_1_5		:=	GVL_IO.b_PWM1_Control_Byte_2 ;
//w_q_677_1_6		:=	GVL_IO.w_PWM1_DO3 ;
//b_q_677_1_7		:=	GVL_IO.b_PWM1_Control_Byte_3
w_q_677_1_8		:=	GVL_IO.w_PWM1_DO4 ;

 b_q_677_2_1		:=	GVL_IO.b_PWM2_Control_Byte_0	;
 w_q_677_2_2		:=	GVL_IO.w_PWM2_DO1;
 w_q_677_2_4		:=	GVL_IO.w_PWM2_DO2;

// _q_1505_1_1	:=	GVL_IO.x_DIG14	;//PTO1
// x_q_1505_1_2	:=	GVL_IO.x_DIG15	;//PTO2
// x_q_1505_1_3	:=	GVL_IO.x_DIG16	;//PTO3
// x_q_1505_1_4	:=	GVL_IO.x_DIG13	;
// x_q_1505_1_5	:=	GVL_IO.x_DIG12	;
// x_q_1505_1_6	:=	GVL_IO.x_DIG01	;
// x_q_1505_1_7	:=	GVL_IO.x_DIG02	;
// x_q_1505_1_8	:=	GVL_IO.x_DIG03	;
// x_q_1505_1_9	:=	GVL_IO.x_DIG04	;
// x_q_1505_1_10	:=	GVL_IO.x_DIG05	;
// x_q_1505_1_11	:=	GVL_IO.x_DIG20	;
// x_q_1505_1_12	:=	GVL_IO.x_DIG24	;
// x_q_1505_1_13	:=	GVL_IO.x_DIG22	;
// x_q_1505_1_14	:=	GVL_IO.x_DIG21	;
// x_q_1505_1_15	:=	GVL_IO.x_DIG25	;
// x_q_1505_1_16	:=	GVL_IO.x_DIG11	;
//
// x_q_1505_2_1	:=	GVL_IO.x_DIG10	;
// x_q_1505_2_2	:=	GVL_IO.x_DIG06	;
// x_q_1505_2_3	:=	GVL_IO.x_DIG17	;
// x_q_1505_2_4	:=	GVL_IO.x_DIG09	;
// x_q_1505_2_5	:=	GVL_IO.x_DIG27	;
// x_q_1505_2_6	:=	GVL_IO.x_DIG23	;
// x_q_1505_2_7	:=	GVL_IO.x_DIG26	;
// x_q_1505_2_8	:=	GVL_IO.x_DIG08	;
// //x_q_1505_2_9	:=	GVL_IO.	;
// x_q_1505_2_10	:=	GVL_IO.x_DIG07	;
// x_q_1505_2_11	:=	GVL_IO.x_DIG19	;
// x_q_1505_2_12	:=	GVL_IO.x_DIG18	;
// //x_q_1505_2_13	:=	GVL_IO.	;
// //x_q_1505_2_14	:=	GVL_IO.	;
// //x_q_1505_2_15	:=	GVL_IO.	;
// //x_q_1505_2_16	:=	GVL_IO.	;
//
// w_q_550_1_1	:=	GVL_IO.w_AI01	;
// w_q_550_1_2	:=	GVL_IO.w_AI02	;
// //w_q_559_1_3	:=	GVL_IO.	;
// //w_q_559_1_4	:=	GVL_IO.	;

(* ---- PLC_PRG.ST ---- *)
PROGRAM PLC_PRG
VAR

	COUNTER : ARRAY[0..7] OF BYTE;
	_FB_InitPeriodicMessage : FB_InitPeriodicMessage;
	//_FB_InitRXMessage : FB_InitRXMessage;
	_GetDateAndTime : dtu.GetDateAndTime;
	_FbModuleConfigurationAndStatus : FbModuleConfigurationAndStatus;
	_FbCanL2Open : FbCanL2Open;
	_FbCanErrorInfo : FbCanErrorInfo;
	_FbCanRx11BitFrameAll : FbCanRx11BitFrameAll;
	_FB_Millis : FB_Millis;
	_FB_RXCanMessageElaboration : FB_RXCanMessageElaboration;
	_FB_handlePeriodicMessages : FB_handlePeriodicMessages;
	msTimer : TON := (IN :=TRUE, PT:= UDINT_TO_TIME(4294967295));
	dtTime : DATE_AND_TIME;
	tActualTime, tLastElapsedTime : TIME;
	stTypFullConfiguration: WagoSysModule_75x_658.typFullConfiguration;
	xCANRxTrigger, xCANdone,xCANbusy,xCANerror,xCAN29BitEnabled,xCANSdoEnabled,xCANDiagOverMbx0Enabled,xCANDiagnosisReset,xCANCommunicationReset: BOOL;
	udiCANBaudrate: udint;
	I_CANport : WagoSysModule_75x_658.I_WagoModule_75x_658Extended;
	eCANBitrate : WagoSysModule_75x_658.eBitrate;
	eCANMode : WagoSysModule_75x_658.eMode := WagoSysModule_75x_658.eMode.CAN_Transparent;
	wCANRxId,wCANCounter:WORD;
	xCANValid,xCANRtrFrame,xCANTriggerResetCounter:BOOL;
	oCANStatus :WagoAppCanLayer2.WagoSysErrorBase.FbResult;
	bCANRxNBytes:BYTE;
	aCANRxBuffer,aCANTxBuffer:ARRAY[1..8]OF BYTE;
	aCANTxBuffer1:ARRAY[0..23]OF BYTE;
	iCanStateMachine, iCANbufferCursor: INT :=0;
	xPeriodicMessageInitDone:BOOL:=FALSE;
	wAliveCounter:WORD;
END_VAR

PLC_INPUT();
PLC_OUTPUT();

IF (NOT xPeriodicMessageInitDone) THEN
	_FB_InitPeriodicMessage(aPeriodicMessages => GVL.aPeriodicMessages);

	I_CANport := CAN_Gateway;
	eCANBitrate := WagoSysModule_75x_658.eBitrate.CAN_500kBits;
	udiCANBaudrate := 500000;
	eCANMode := WagoSysModule_75x_658.eMode.CAN_Transparent;
	xCAN29BitEnabled := FALSE;
	xCANSdoEnabled := FALSE;
	xCANDiagOverMbx0Enabled := FALSE;
	xCANCommunicationReset := FALSE;

	xPeriodicMessageInitDone := TRUE;
	//_FB_InitRXMessage(aRXMessages => gvl.aRXMessages);
END_IF

_GetDateAndTime(xExecute := TRUE,
				dtDateAndTime => dtTime
				);
msTimer();
tActualTime := msTimer.ET;

CASE iCanStateMachine OF
	0: //write config values
		_FbModuleConfigurationAndStatus(I_Port := I_CANport,
										xExecute := TRUE,
										xWriteRead := FALSE,//NOT xCANdone,
										xSaveValues := TRUE,
										dtTime := dtTime,
										eBitrate := eCANBitrate,
										eMode := eCANMode,
										x29BitEnabled := xCAN29BitEnabled,
										xSdoEnabled := xCANSdoEnabled,
										xDiagOverMbx0Enabled := xCANDiagOverMbx0Enabled,
										typConfigData := stTypFullConfiguration,
										xDiagnosisReset := xCANDiagnosisReset,
										xCommunicationReset := xCANCommunicationReset,
										xCheckConfiguration := TRUE,
										xDone => xCANdone,
										xBusy => xCANbusy,
										xError => xCANerror,
										oStatus =>oCANStatus,
										xDataMatches =>,
										eDiagnosisErrorCode =>,
										bDiagnosisChannelNo =>,
										eDiagnosisMode =>,
										eDiagnosisType =>,
										wDiagnosisErrorCounter =>,
										wDiagnosisWarningCounter =>,
										wDiagnosisTotalCounter =>,
										xStatusBitModulError =>,
										xStatusBitRxOverflow =>,
										xStatusBitRxOverflow =>,
										xStatusBitCanError =>
										);

		IF _FbModuleConfigurationAndStatus.xDone AND NOT _FbModuleConfigurationAndStatus.xError THEN
			iCanStateMachine := 1;
		ELSIF _FbModuleConfigurationAndStatus.xError THEN
			iCanStateMachine := 99;
		END_IF

	1: //look for errors
		_FbCanErrorInfo(xEnable:= TRUE,
						I_Port := I_CANport,
						xTriggerResetCounter := xCANTriggerResetCounter,
						xValid=>,
						xError=>,
						oStatus=>,
						wBusState=>,
						wBusDiag=>);

		IF _FbCanErrorInfo.xValid AND NOT _FbCanErrorInfo.xError THEN
			iCanStateMachine := 2;
		ELSIF _FbCanErrorInfo.xError THEN
			iCanStateMachine := 99;
		END_IF

	2: //open can layer2 port + RX + TX
		_FbModuleConfigurationAndStatus(I_Port := I_CANport,
								xExecute := TRUE,
								xWriteRead := FALSE,//NOT xCANdone,
								xSaveValues := FALSE,
								dtTime := dtTime,
								eBitrate := eCANBitrate,
								eMode := eCANMode,
								x29BitEnabled := xCAN29BitEnabled,
								xSdoEnabled := xCANSdoEnabled,
								xDiagOverMbx0Enabled := xCANDiagOverMbx0Enabled,
								typConfigData := stTypFullConfiguration,
								xDiagnosisReset := xCANDiagnosisReset,
								xCommunicationReset := xCANCommunicationReset,
								xCheckConfiguration := TRUE,
								xDone => ,
								xBusy => ,
								xError => ,
								oStatus =>,
								xDataMatches =>,
								eDiagnosisErrorCode =>,
								bDiagnosisChannelNo =>,
								eDiagnosisMode =>,
								eDiagnosisType =>,
								wDiagnosisErrorCounter =>,
								wDiagnosisWarningCounter =>,
								wDiagnosisTotalCounter =>,
								xStatusBitModulError =>,
								xStatusBitRxOverflow =>,
								xStatusBitRxOverflow =>,
								xStatusBitCanError =>
								);

		_FbCanL2Open(xEnable:= TRUE,
						I_Port := I_CANport,
						udiBaudrate := udiCANBaudrate,
						dwFlags := 0,
						dwpara := 0);

		IF _FbModuleConfigurationAndStatus.xDone AND NOT _FbModuleConfigurationAndStatus.xError THEN
			xCANRxTrigger := TRUE;
			_FbCanRx11BitFrameAll(	xEnable := _FbModuleConfigurationAndStatus.xDone,
									I_Port := I_CANport,
									xBufferMode := TRUE,
									xRxTrigger := xCANRxTrigger,
									xValid => xCANValid,
									xError => xCANError,
									xBusy => xCANBusy,
									oStatus => oCANStatus,
									wCounter => ,
									xRtrFrame => xCANRtrFrame,
									bRxNBytes => bCANRxNBytes,
									aRxBuffer => ,
									wRxId => wCANRxId);
		END_IF

		//RECEIVED MESSAGES
		IF _FbCanRx11BitFrameAll.xValid AND (_FbCanRx11BitFrameAll.wFrames>0) THEN
			//more than one message received
			FOR iCANbufferCursor := 1 TO WORD_TO_INT(_FbCanRx11BitFrameAll.wFrames) DO

				_FB_RXCanMessageElaboration(wRxId := DWORD_TO_WORD(_FbCanRx11BitFrameAll.auxRxData[iCANbufferCursor].dwID),
									bRxNBytes := _FbCanRx11BitFrameAll.auxRxData[iCANbufferCursor].bLen,
									aRxBuffer := _FbCanRx11BitFrameAll.auxRxData[iCANbufferCursor].aData
									);
			END_FOR
			wCANCounter := _FbCanRx11BitFrameAll.wCounter;
		ELSIF  _FbCanRx11BitFrameAll.xValid AND (_FbCanRx11BitFrameAll.wFrames = 0) AND (_FbCanRx11BitFrameAll.wCounter>wCANCounter) THEN
			//only one message received
			_FB_RXCanMessageElaboration(wRxId := _FbCanRx11BitFrameAll.wRxId,
								bRxNBytes := _FbCanRx11BitFrameAll.bRxNBytes,
								aRxBuffer := _FbCanRx11BitFrameAll.aRxBuffer
								);
			wCANCounter := _FbCanRx11BitFrameAll.wCounter;
		ELSIF _FbCanRx11BitFrameAll.xError OR _FbModuleConfigurationAndStatus.xError THEN
			iCanStateMachine := 99;
		END_IF

		//TRANSMITTED MESSAGES: periodic
		FOR iCANbufferCursor:=1 TO GVL.uiPeriodcMessageN DO
			mem.MemFill(pMemoryBlock := ADR(aCANTxBuffer),
						uiLength := SIZEOF(aCANTxBuffer),
						byfillvalue :=0);

			CASE iCANbufferCursor OF
				//insert here the data field of the message
				1:  //BANCO_VCM4_Alive
					IF wAliveCounter<65535 THEN
						wAliveCounter := wAliveCounter + 1;
					ELSE
						wAliveCounter := 0;
					END_IF
					aCANTxBuffer[1] := WORD_TO_BYTE(SHR(wAliveCounter,8));
					aCANTxBuffer[2] := WORD_TO_BYTE(wAliveCounter);

				2: 	//BANCO_VCM4_DOUT

					aCANTxBuffer[1].0 := GVL_IO.x_DOV01;
					aCANTxBuffer[1].1 := GVL_IO.x_DOV02;
					aCANTxBuffer[1].2 := GVL_IO.x_DOV03;
					aCANTxBuffer[1].3 := GVL_IO.x_DOV04;
					aCANTxBuffer[1].4 := GVL_IO.x_DOV05;
					aCANTxBuffer[1].5 := GVL_IO.x_DOV06;
					aCANTxBuffer[1].6 := GVL_IO.x_DOV07;
					aCANTxBuffer[1].7 := GVL_IO.x_DOV08;
					aCANTxBuffer[2].0 := GVL_IO.x_DOG01;
					aCANTxBuffer[2].1 := GVL_IO.x_DOG02;
					aCANTxBuffer[2].2 := GVL_IO.x_DOG03;
					aCANTxBuffer[2].3 := GVL_IO.x_DOG04;
					aCANTxBuffer[2].4 := GVL_IO.x_DOG05;
					aCANTxBuffer[2].5 := GVL_IO.x_DOG06;
					aCANTxBuffer[2].6 := GVL_IO.x_DOG07;
					aCANTxBuffer[3].0 := GVL_IO.x_DOG08;
					aCANTxBuffer[3].1 := GVL_IO.x_DOG09;
					aCANTxBuffer[3].2 := GVL_IO.x_DOG10;
					aCANTxBuffer[3].3 := GVL_IO.x_DOG11;
					aCANTxBuffer[3].4 := GVL_IO.x_DOG12;
			END_CASE

			_FB_handlePeriodicMessages( tActualTime := tActualTime,
										tLastElapsedTime := GVL.aPeriodicMessages[iCANbufferCursor].tLastElapsedTime,
										tPeriod := GVL.aPeriodicMessages[iCANbufferCursor].tPeriod,
										wTxId := GVL.aPeriodicMessages[iCANbufferCursor].wTxId,
										bTxNBytes := GVL.aPeriodicMessages[iCANbufferCursor].bTxNBytes,
										aTxBuffer := aCANTxBuffer,
										);

			aCANTxBuffer1[0] := 1;
			aCANTxBuffer1[1] := 2;
			aCANTxBuffer1[2] := 3;
			aCANTxBuffer1[3] := 4;
			aCANTxBuffer1[4] := 5;
			aCANTxBuffer1[5] := 6;
			aCANTxBuffer1[6] := 7;
			aCANTxBuffer1[7] := 8;

// 			GVL_IO.w_CAN_SEND[0] := aCANTxBuffer1[0];
// 			GVL_IO.w_CAN_SEND[1] := aCANTxBuffer1[1];
// 			GVL_IO.w_CAN_SEND[2] := aCANTxBuffer1[2];
// 			GVL_IO.w_CAN_SEND[3] := aCANTxBuffer1[3];
// 			GVL_IO.w_CAN_SEND[4] := aCANTxBuffer1[4];
// 			GVL_IO.w_CAN_SEND[5] := aCANTxBuffer1[5];
// 			GVL_IO.w_CAN_SEND[6] := aCANTxBuffer1[6];
// 			GVL_IO.w_CAN_SEND[7] := aCANTxBuffer1[7];

// 			_FB_handlePeriodicMessages( tActualTime := tActualTime,
// 										tLastElapsedTime := GVL.aPeriodicMessages[iCANbufferCursor].tLastElapsedTime,
// 										tPeriod := GVL.aPeriodicMessages[iCANbufferCursor].tPeriod,
// 										wTxId := GVL.aPeriodicMessages[iCANbufferCursor].wTxId,
// 										bTxNBytes := GVL.aPeriodicMessages[iCANbufferCursor].bTxNBytes,
// 										aTxBuffer := aCANTxBuffer1,
// 										);

		END_FOR
	99: //error --> retry
		iCanStateMachine := 2;
		//GVL_IO.x_DHLC01 := TRUE;

END_CASE
